Universal Robots PolyScope program: xmlrpc_deteccion_fresas_vertical.urp

Program xmlrpc_deteccion_fresas_vertical (installation=deteccion_fresas directory=/programs/usbdisk/Versiones xmlrpc_deteccion_fresas createdIn=5.17.0 lastSavedIn=5.21.3 robotSerialNumber=20185300103)
Calibrated DH parameters: a=[-0.00011, -0.177742, -0.140941, 0.000115, -0.000132, 0]; d=[0.151657, 34.818115, -45.396006, 10.707357, 0.085307, 0.091775]; alpha=[1.570734, 0.004798, -0.015068, 1.570708, -1.571204, 0]; deltaTheta=[0, 0.754463, 0.092237, -0.846764, -0.000014, 0]
InitVariablesNode
BeforeStart
  Folder Configuracion XMLRPC
    'Configuración del XMLRPC'
    camera := rpc_factory("xmlrpc","http://192.168.23.107:50000")
  Folder Inicializacipn variables
    'Variable para ver si se detecta dos veces el mismo pto'
    next_pose_aux := p[0,0,0,0,0,0]
  Folder Centro coord camara
    'Punto de referencia de la camara (centro de coordenadas camara)'
    SuppressedNode
      MoveJ speed 60 deg/s, acceleration 80 deg/s^2 (useActiveTCP=true optimoveEnabled=false optiMoveSpeed=0.3 optiMoveAcceleration=0.09) feature=Plano_camara
        Waypoint reference_p: TCP in base x=-205.136 y=303.641 z=-13.102 mm, rx=-1.1967 ry=-2.9046 rz=-0.0001 rad; joints [-215.195, -141.895, -109.787, -18.283, 89.252, -81.03] deg; TCP offset x=0 y=0 z=20 mm, rx=0 ry=0 rz=0 rad; feature pose in base x=-205.136 y=303.641 z=-13.102 mm, rx=-1.1967 ry=-2.9046 rz=-0.0001 rad
Robot Program (runOnlyOnce=false)
  Folder Home
    'Home: Punto inicial para posterior recogida de deteccion'
    MoveJ speed 60 deg/s, acceleration 80 deg/s^2 (useActiveTCP=true optimoveEnabled=true optiMoveSpeed=0.21 optiMoveAcceleration=0.044) feature=Plano_pared
      Waypoint Casa: TCP in base x=78.353 y=-233.897 z=362.624 mm, rx=-0.7295 ry=1.7607 rz=-1.6169 rad; joints [310.596, -27.266, -145.549, -10, 98.288, 3.553] deg; TCP offset x=0 y=0 z=140 mm, rx=0 ry=0 rz=0 rad; feature pose in base x=17.54 y=-260.336 z=444.744 mm, rx=-0.673 ry=1.7392 rz=-1.7253 rad
  Folder Comunicacion camara
    'Obtencion de datos de la camara'
    next_pose := camera.get_next_pose()
    'Se hace el cambio de unidades mm a m'
    next_pose_list := p[next_pose[0]/1000,next_pose[1]/1000,0,0,0,0]
  Folder Movimiento UR
    If next_pose_list[0]≟0  and next_pose_list[1]≟0
      Folder NO_Deteccion
        MoveJ speed 60 deg/s, acceleration 80 deg/s^2 (useActiveTCP=true optimoveEnabled=false optiMoveSpeed=0.3 optiMoveAcceleration=0.09) feature=Plano_pared
          Waypoint Casa: TCP in base x=78.353 y=-233.897 z=362.624 mm, rx=-0.7295 ry=1.7607 rz=-1.6169 rad; joints [310.596, -27.266, -145.549, -10, 98.288, 3.553] deg
    Else 
      Folder Deteccion_OK
        If next_pose_aux ≠ next_pose_list
          'Hay detecciones que recoger'
          'Posicion de la recogida'
          MoveL speed 250 mm/s, acceleration 1200 mm/s^2 (useActiveTCP=true optimoveEnabled=false optiMoveSpeed=0.3 optiMoveAcceleration=0.09) feature=Plano_pared
            Waypoint Variable (Variable): variable=next_pose_list
          'Variable aux para comparar listas '
          next_pose_aux := p[next_pose_list[0],next_pose_list[1],next_pose_list[2],0,0,0]
        Else 
          'No hay detecciones que recoger'
          MoveJ speed 60 deg/s, acceleration 80 deg/s^2 (useActiveTCP=true optimoveEnabled=false optiMoveSpeed=0.3 optiMoveAcceleration=0.09) feature=Plano_pared
            Waypoint Casa: TCP in base x=78.353 y=-233.897 z=362.624 mm, rx=-0.7295 ry=1.7607 rz=-1.6169 rad; joints [310.596, -27.266, -145.549, -10, 98.288, 3.553] deg
  Wait Sleep waitTime=1
